{attribute 'obsolete' := 'EL5042_Status has been renamed to ST_EL5042_Status'}
TYPE EL5042_Status : ST_EL5042_Status; END_TYPE

(* stored: Version 1.1.0.1
   DUT EL5042_Status: Id {8d65cae0-9efe-4c5b-a7a7-f17022f98dd4} *)
